{attribute 'GeneratedUsingTerminal: EP1816-3008-0016'}
{attribute addProperty BoxType "EP1816-3008-0016"}
{attribute addProperty Id "StatusAT %I*Status_A3AA621F2ValueAT %I*INT2"}
{attribute addProperty CRC "3286137354"}
{attribute addProperty Size "4"}
TYPE AI_Inputs_Channel_C3DE7A0A :
STRUCT
	{attribute addProperty Name "Status"}
	Status AT %I* : Status_A3AA621F;
	{attribute addProperty Name "Value"}
	Value AT %I* : INT;
END_STRUCT
END_TYPE

(* stored: Version 1.2.0.0, ProductVersion 3.1.4024.9
   DUT AI_Inputs_Channel_C3DE7A0A: Id {1fbf9adb-bc7f-48c5-8df2-7dce41984679} *)
